(* Schneider Machine Expert - Basic project motor_start_stop_TM221CE24T, file version 3.0.0.0 *)
(* ProjectInformations: Name=Motor Start Stop TM221CE24T *)

HARDWARE
  Cpu 0: TM221CE24T
  EthernetConfiguration: NetworkName=M221, IpAllocationMode=ByDhcp, IpAddress=192.168.1.10, SubnetMask=255.255.255.0
  SerialLineConfiguration: Baud=Baud19200, Parity=ParityEven, DataBits=DataBits8, StopBits=StopBits1, PhysicalMedium=PhysicalMediumRs485, TransmissionMode=TransmissionModeModbusRtu, SlaveId=1, Addressing=SlaveAddressing
  MastTask: UsePeriodScanMode=false, PeriodScan=100
  FastTask: Period=255
  CpuBehavior: StartingMode=StartAsPreviousState, AutoSaveRamOnEeprom=true, WatchdogPeriod=250

SYMBOLS  (address, symbol, comment, settings)
  %I0.0     START_MOTOR
  %I0.1     STOP_MOTOR
  %I0.2     ESTOP
  %I0.3     OVERLOAD
  %Q0.0     MOTOR_RUN
  %Q0.1     ALARM

POU Motor Control
  (* SectionNumber=1 *)

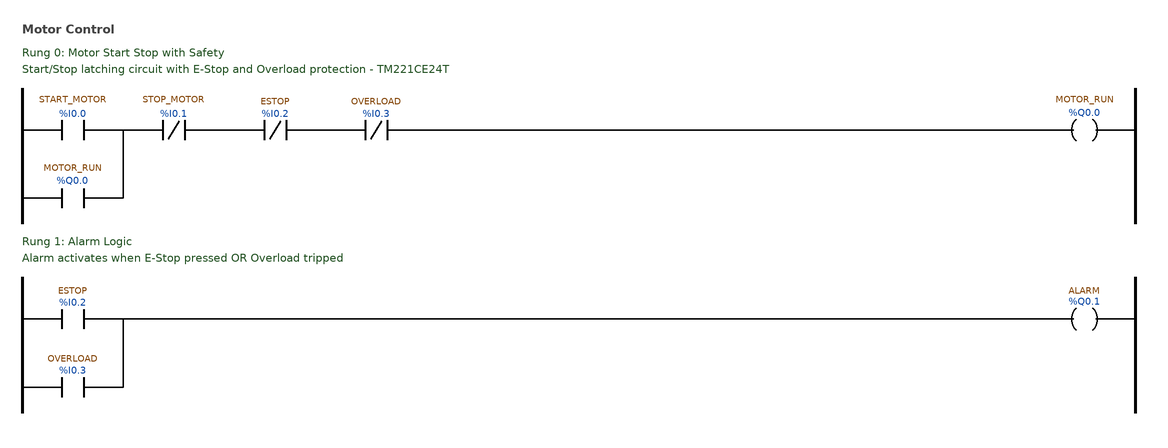

// Rung 0: Motor Start Stop with Safety
// Start/Stop latching circuit with E-Stop and Overload protection - TM221CE24T
  LD %I0.0                (* START_MOTOR *)
  OR %Q0.0                (* MOTOR_RUN *)
  ANDN %I0.1              (* STOP_MOTOR *)
  ANDN %I0.2              (* ESTOP *)
  ANDN %I0.3              (* OVERLOAD *)
  ST %Q0.0                (* MOTOR_RUN *)
  // as ST:
  //   MOTOR_RUN := (START_MOTOR OR MOTOR_RUN) AND NOT STOP_MOTOR AND NOT ESTOP AND NOT OVERLOAD;

// Rung 1: Alarm Logic
// Alarm activates when E-Stop pressed OR Overload tripped
  LD %I0.2                (* ESTOP *)
  OR %I0.3                (* OVERLOAD *)
  ST %Q0.1                (* ALARM *)
  // as ST:
  //   ALARM := ESTOP OR OVERLOAD;
